FUNCTION_BLOCK FB_WashingMachine
VAR

    // ── State ────────────────────────────────────────── 
    eState      : E_WashState := E_WashState.IDLE; 
    bStateEntry : BOOL        := TRUE; 
    // ── Strategy (interface reference — DIP) ─────────── 
    ipGetStrategy   : I_WashStrategy; 
    bStrategySet : BOOL := FALSE; 
    // ── Cached settings from strategy ───────────────── 
    stWashSettings  : ST_WashSettings; 
    // ── Control flags ───────────────────────────────── 
   bDoorLocked : BOOL := FALSE; 
    bRunning    : BOOL := FALSE; 
 // ── Monitoring / Log ────────────────────────────── 
    sLog      : STRING; 
    sErrorMessage : STRING; 
// ── Timers ──────────────────────────────────────── 
    fbOnState     : TON;   // Drives each timed state 
    fbOnCompleted : TON;   // Auto-return COMPLETED → IDLE 

	
END_VAR

// ── Cyclic timers ──────────────────────────────────────── 

fbOnState    (IN := bRunning, PT := stWashSettings.tWashDuration); 
fbOnCompleted(IN := (eState = E_WashState.COMPLETED),  PT := GVL_WashConstants.COMPLETED_HOLD_TIME); 


CASE eState OF 
  E_WashState.IDLE: 
    IF bStateEntry THEN 
        bRunning    := FALSE; 
        bDoorLocked := FALSE; 
        sLog        := 'STATE: IDLE — Select program and press Start.'; 
        bStateEntry := FALSE; 
    END_IF 

  E_WashState.FILLING:                         // NEW STATE 
    IF bStateEntry THEN 
        fbOnState(IN := FALSE, PT := GVL_WashConstants.FILL_TIME); 
        fbOnState(IN := TRUE,  PT := GVL_WashConstants.FILL_TIME); 
        sLog        := 'STATE: FILLING — Drum filling with water.'; 
        bStateEntry := FALSE; 
    END_IF 

    fbOnState(IN := TRUE, PT := GVL_WashConstants.FILL_TIME); 
    IF fbOnState.Q THEN 
        sLog := 'TRANSITION: FILLING → WASHING'; 
        GoTo(E_WashState.WASHING); 
    END_IF 

  E_WashState.WASHING: 
    IF bStateEntry THEN 
        fbOnState(IN := FALSE, PT := stWashSettings.tWashDuration); 
        fbOnState(IN := TRUE,  PT := stWashSettings.tWashDuration); 
        sLog := CONCAT('STATE: WASHING — Program: ', 
                  CONCAT(ipGetStrategy.GetProgramName(), 
                  CONCAT(' | Temp: ', 
                  CONCAT(REAL_TO_STRING(stWashSettings.rTemperature), 'C')))); 
        bStateEntry := FALSE; 
    END_IF 

    fbOnState(IN := TRUE, PT := stWashSettings.tWashDuration); 
    IF fbOnState.Q THEN 
        sLog := 'TRANSITION: WASHING → DRAINING'; 
        GoTo(E_WashState.DRAINING); 
    END_IF 

  E_WashState.DRAINING:                        // NEW STATE 
    IF bStateEntry THEN 
        fbOnState(IN := FALSE, PT := GVL_WashConstants.DRAIN_TIME); 
        fbOnState(IN := TRUE,  PT := GVL_WashConstants.DRAIN_TIME); 
        sLog        := 'STATE: DRAINING — Emptying drum.'; 
        bStateEntry := FALSE; 
    END_IF 

    fbOnState(IN := TRUE, PT := GVL_WashConstants.DRAIN_TIME); 
    IF fbOnState.Q THEN 
        sLog := 'TRANSITION: DRAINING → COMPLETED'; 
        GoTo(E_WashState.COMPLETED); 
    END_IF 

  E_WashState.COMPLETED: 
    IF bStateEntry THEN 
        bRunning    := FALSE; 
        sLog        := 'STATE: COMPLETED — Cycle done. Door unlocking soon.'; 
        bStateEntry := FALSE; 
    END_IF 

    fbOnCompleted(IN := TRUE, PT := GVL_WashConstants.COMPLETED_HOLD_TIME); 

    IF fbOnCompleted.Q THEN 
        sLog := 'TRANSITION: COMPLETED → IDLE'; 
        GoTo(E_WashState.IDLE); 
    END_IF 

  E_WashState.ERROR: 
    IF bStateEntry THEN 
        bRunning    := FALSE; 
        bDoorLocked := FALSE; 
        sLog        := CONCAT('STATE: ERROR — ', sErrorMessage); 
        bStateEntry := FALSE; 
    END_IF  // Cleared only via ResetError() 
  ELSE 

    GoTo(E_WashState.IDLE); 
END_CASE

PROPERTY CurrentState : E_WashState
GET
VAR
	eCurrentState: E_WashState;
END_VAR
 CurrentState := eState;
END_GET
SET
END_SET
END_PROPERTY

PROPERTY ErrorMessage : STRING
GET

    ErrorMessage := sErrorMessage;
END_GET
SET
END_SET
END_PROPERTY

METHOD PRIVATE GoTo : BOOL
VAR_INPUT 
eNext : E_WashState;
 END_VAR

 eState := eNext;
 bStateEntry := TRUE;
END_METHOD

PROPERTY IsRunning : BOOL
GET

    IsRunning := bRunning;
END_GET
SET
END_SET
END_PROPERTY

METHOD LockDoor : BOOL
VAR_INPUT
END_VAR
 IF eState <> E_WashState.IDLE THEN 

        sLog := 'ERROR: Door lock only from IDLE.'; LockDoor := FALSE; RETURN; 

    END_IF 

    bDoorLocked := TRUE; 
sLog := 'Door LOCKED.'; 
LockDoor := TRUE;
END_METHOD

PROPERTY LogMessage : STRING
GET

    LogMessage := sLog;
END_GET
SET
END_SET
END_PROPERTY

PROPERTY  RemainingTime : TIME
GET
 IF fbOnState.PT > fbOnState.ET THEN
        RemainingTime := fbOnState.PT - fbOnState.ET; 
    ELSE 
     RemainingTime := T#0S; 
    END_IF
END_GET
SET
END_SET
END_PROPERTY

METHOD ResetError : BOOL
VAR_INPUT
END_VAR
IF eState <> E_WashState.ERROR THEN 
       sLog := 'RESET: Not in ERROR.'; ResetError := FALSE; RETURN; 
    END_IF 
	
    sErrorMessage    := ''; 
    bStrategySet := FALSE; 
    sLog         := 'RESET: Error cleared. Select program and restart.'; 
    GoTo(E_WashState.IDLE);
    ResetError := TRUE;
END_METHOD

METHOD  SelectStrategy : BOOL

VAR_INPUT 
    ipStrategy : I_WashStrategy; 
END_VAR
IF bRunning THEN 
       sLog := 'ERROR: Cannot change program while running.';
        SelectStrategy := FALSE; RETURN; 
    END_IF 

    IF ipStrategy = 0 THEN 
        sLog := 'ERROR: Invalid strategy reference.'; 
        SelectStrategy := FALSE; RETURN;
    END_IF 

    ipGetStrategy   := ipStrategy; 
    stWashSettings   := ipGetStrategy.GetSettings(); 
    bStrategySet := TRUE; 
    // Validate temperature 

    IF stWashSettings.rTemperature > GVL_WashConstants.TEMP_MAX OR 
       stWashSettings.rTemperature < GVL_WashConstants.TEMP_MIN THEN 
        sErrorMessage := 'Temperature out of safe range'; 
        GoTo(E_WashState.ERROR); SelectStrategy := FALSE; RETURN; 
    END_IF 

    // Validate spin speed 

    IF stWashSettings.nSpinSpeed > GVL_WashConstants.SPIN_MAX OR 
      stWashSettings.nSpinSpeed < GVL_WashConstants.SPIN_MIN THEN 
        sErrorMessage := 'Spin speed out of safe range'; 
        GoTo(E_WashState.ERROR); SelectStrategy := FALSE; RETURN; 
    END_IF 

    ipGetStrategy.Start();   // Call strategy Start() per interface contract 
    sLog          := CONCAT('Program selected: ', ipGetStrategy.GetProgramName()); 
    SelectStrategy := TRUE;
END_METHOD

METHOD  Start : BOOL
VAR_INPUT
END_VAR
IF eState <> E_WashState.IDLE THEN 
        sLog := 'ERROR: Not in IDLE.'; Start := FALSE; RETURN; 
    END_IF 
	
    IF NOT bStrategySet OR ipGetStrategy = 0 THEN 
        sLog := 'ERROR: No program selected.'; Start := FALSE; RETURN; 
    END_IF 
	
    IF NOT bDoorLocked THEN 
        sLog := 'ERROR: Door not locked.'; Start := FALSE; RETURN; 
    END_IF 

    bRunning := TRUE; 
    sLog     := CONCAT('START: ', ipGetStrategy.GetProgramName()); 
    GoTo(E_WashState.FILLING);   // First state is now FILLING 
    Start     := TRUE;
END_METHOD

METHOD  Stop : BOOL
VAR_INPUT
END_VAR

// Edge case — already idle
    IF NOT bRunning THEN 
       sLog := 'STOP: Not running.'; RETURN; 
   END_IF 
    sErrorMessage := 'Cycle stopped by operator'; 
    GoTo(E_WashState.ERROR);
END_METHOD

PROPERTY WashDuration : TIME
GET
   IF bStrategySet AND ipGetStrategy <> 0 THEN
        WashDuration := ipGetStrategy.GetDuration();
    ELSE
        WashDuration := T#0S;
    END_IF
END_GET
SET
END_SET
END_PROPERTY

END_FUNCTION_BLOCK

(* stored: Version 1.1.0.1, ProductVersion 3.1.4024.16
   POU FB_WashingMachine: Id {182d94af-703d-4404-b9f5-16db70894ffa}, SpecialFunc None
   Property CurrentState: Id {d69cb94e-a7b2-4bd0-9661-5e10d0a1df2b}
   Get Get: Id {3fc6311a-f53f-4bce-a7c2-3e8078fa9d41}
   Set Set: Id {097f0d05-d0e7-4c3a-aad4-5670303745e2}
   Property ErrorMessage: Id {855ecaa8-948b-46a2-81bb-097035a257c1}
   Get Get: Id {8387c281-0323-48c5-a7c1-7900485f94af}
   Set Set: Id {2afaca2f-d3dc-4310-b7e2-31172879f092}
   Method GoTo: Id {0d6ddf0b-eea5-4757-815f-acba3a290d2f}
   Property IsRunning: Id {05ce31fd-bba2-439b-a2ae-6ff6e930fec9}
   Get Get: Id {6ec5ce81-8d8a-4cb2-a657-4f8c749c0e28}
   Set Set: Id {30254e30-a4d2-4e57-9824-9ea3d28be941}
   Method LockDoor: Id {e3177fec-6683-41aa-94f6-9d039fb67bd4}
   Property LogMessage: Id {e9542b3e-00d9-4d10-8acc-dad4ea2fc7b9}
   Get Get: Id {0cc44213-e29f-46d7-b2b0-0d2e31cf18d4}
   Set Set: Id {882225c5-3cba-457f-942a-e086df3ee95f}
   Property RemainingTime: Id {3e393044-01f3-4c2b-b907-f51eed3a5a8e}
   Get Get: Id {57aa9742-0208-4dd7-9579-c7f79b9e0560}
   Set Set: Id {7de6a2ec-98fc-4124-952c-9819ccee5d24}
   Method ResetError: Id {6eb0be3c-ae30-46d6-bc3f-446ce0a650d5}
   Method SelectStrategy: Id {11f9c0a5-9ac0-443b-9068-0c6940a261ee}
   Method Start: Id {2d973bb1-1019-4bf5-b0f1-6f99297b2521}
   Method Stop: Id {1c3be39f-7ad2-40d8-b663-0a6b75deae94}
   Property WashDuration: Id {94ebbba6-10d1-4fb1-b3fe-8a14774ccaa3}
   Get Get: Id {3ff4800e-bf6c-4d5e-ae3e-6baa3b76ca66}
   Set Set: Id {66c8d3f3-e5b6-466a-b023-197b4efad9aa} *)
